/// calibration that is determined by calibration sequences of the unit (static offsets, shifts)
TYPE TransportDataCalibration :
STRUCT
END_STRUCT
END_TYPE

(* stored: Version 1.1.0.1
   DUT TransportDataCalibration: Id {a1fd903c-250a-4a1c-a1a3-9f7fa5b5ea5a} *)
